(* CoDeSys 2.3.9.50 project: AXIS_CONTROL.pro *)
(* Libraries: TcBase.lib 14.5.09 12:14:08, TcSystem.lib 7.6.16 11:01:22, TcBaseMath.lib 27.7.04 12:07:56, TcMath.lib 23.9.04 15:15:30, TcNC.lib 10.10.08 17:55:34, TcUtilities.lib 3.2.16 16:08:58, TcEtherCAT.lib 30.11.16 19:52:18, TcTestAndSet.lib 23.2.09 12:50:08, TcDrive.lib 25.1.17 09:42:28, TcMc2Drive.lib 19.1.10 11:34:38, TcMC2.lib 19.10.15 15:49:44, STANDARD.LIB 5.6.98 12:03:02 *)

(* Task configuration *)
TASK Standard (PRIORITY := 0, INTERVAL := T#1ms);
	MAIN
END_TASK

(* Global variable list: Global_Variables_Hardware *)
VAR_GLOBAL

	input : STRING(35):='';
	Unit: REAL;
(*motor x*)
	fbNcAxis_Axis_X	: FB_NcAxis;
	stAxis_X			: ST_NcAxis;
	Axis_x			: AXIS_REF;


(*motor y*)
	fbNcAxis_Axis_Y	: FB_NcAxis;
	stAxis_Y			: ST_NcAxis;
	Axis_y			: AXIS_REF;

	Axis_dummy	: AXIS_REF;
END_VAR

(* Global variable list: TwinCAT_Configuration *)
(* Generated automatically by TwinCAT - (read only) *)
VAR_CONFIG
	.Axis_x.PlcToNc AT %QB0 : PLCTONC_AXIS_REF;	(*  ~ {LinkedWith:TINC^NC-Task 1 SAF^Axes^Axis 1^Inputs^Axis 1_FromPlc} *)
	.Axis_x.NcToPlc AT %IB0 : NCTOPLC_AXIS_REF;	(*  ~ {LinkedWith:TINC^NC-Task 1 SAF^Axes^Axis 1^Outputs^Axis 1_ToPlc} *)
	.Axis_y.PlcToNc AT %QB128 : PLCTONC_AXIS_REF;	(*  ~ {LinkedWith:TINC^NC-Task 1 SAF^Axes^Axis 2^Inputs^Axis 2_FromPlc} *)
	.Axis_y.NcToPlc AT %IB128 : NCTOPLC_AXIS_REF;	(*  ~ {LinkedWith:TINC^NC-Task 1 SAF^Axes^Axis 2^Outputs^Axis 2_ToPlc} *)
	.Axis_dummy.PlcToNc AT %QB256 : PLCTONC_AXIS_REF;
	.Axis_dummy.NcToPlc AT %IB256 : NCTOPLC_AXIS_REF;
END_VAR

(* Data type in DataTypes/FBsTypes/NC_Axis_Params/AxisVariables *)
TYPE ST_AxisVars :
STRUCT
	ax_ctrl:ST_ctrl;
	ax_stat:ST_stat;
END_STRUCT
END_TYPE

(* Data type in DataTypes/FBsTypes/NC_Axis_Params/AxisVariables *)
TYPE ST_ctrl :
STRUCT

(*ReadNCParam*)
	ReadParamExe:BOOL;
	ReadParamNum: mc_axisparameter:=AxisEncoderModuloValue;

(*Pwr,Reset*)
	Enable:BOOL;
	Enable_inhibit:BOOL;
	En_FW:BOOL;
	En_BW:BOOL;
	Reset:BOOL;
	Override:REAL:=100;
(*Stop*)
	StopExe:BOOL;
	StopDec:REAL;
(*SetPosition*)
	SetPosExe:BOOL;
	SetPosition:REAL;
(*Homing*)
	HomeExe:BOOL;
	HomeSW: BOOL;
	LimitSW_Max:BOOL;
	LimitSW_Min:BOOL;
	HomeSetPos:REAL;
	HomeOffsetPos:REAL;
	HomeOffsetVelo:REAL:=1;
(*Jog*)
	JogFW:BOOL;
	JogBW:BOOL;
	JogVel:REAL:=1;
	JogAcc:REAL;
	JogDec:REAL;
	JogMode: E_JogMode:=MC_JOGMODE_CONTINOUS;
(*MoveRelative*)
	MrelExe:BOOL;
	MrelDist:REAL;
	MrelVel:REAL:=1;
	MrelAcc:REAL;
	MrelDec:REAL;
(*MoveAbsolute*)
	MabsExe:BOOL;
	MabsPos:REAL;
	MabsVel:REAL:=1;
	MabsAcc:REAL;
	MabsDec:REAL;
	MabsBufferMode:MC_BufferMode;
(*MoveAbsoluteBlending*)
	MabsBlendExe:BOOL;
	MabsBlendPos:REAL;
	MabsBlendVel:REAL:=1;
	MabsBlendAcc:REAL;
	MabsBlendDec:REAL;
	MabsBlendBufferMode:MC_BufferMode;
(*MoveModulo*)
	MmodExe:BOOL;
	MmodPos:REAL;
	MmodVel:REAL:=1;
	MmodAcc:REAL;
	MmodDec:REAL;
	MmodDir:MC_Direction :=MC_Positive_Direction;(*MC_Positive_Direction := 1,MC_Shortest_Way ,MC_Negative_Direction ,  MC_Current_Direction *)
(*MoveVelocity*)
	MvelExe:BOOL;
	MvelVelo:REAL:=1;
	MvelAcc:REAL;
	MvelDec:REAL;
	MvelDirection:MC_Direction ;
	MvelPStopEnable:BOOL;
	MvelPStopPos:REAL;
	MvelPStopAcc:REAL;
	MvelPStopDec:REAL;
(*GearingDyn*)
	GrInDynExe:BOOL;
	GearRatio:REAL;
	GrInAcc:REAL;
	GrInDec:REAL;
	GearOut:BOOL;
(*GearingMultimaster*)
	GrInMMstrExe:BOOL;
	GearRatioMstr:REAL;
	GearRatioMstr2:REAL;
	GearRatioMstr3:REAL;
	GearRatioMstr4:REAL;
	GrInMMstrAcc:REAL;
	GrInMMstrDec:REAL;
	GearMMstrOut:BOOL;
(*TouchProbe*)
	TriggerRef : trigger_ref;
	TProbeExe:BOOL;
	TPWindowOnly: BOOL;
	TPFirstPosition:REAL;
	TPLastPosition :REAL;
(*AbortTouchProbe*)
	AbortTrigger:BOOL;
(*MoveSuperimposed*)
	SImpExe : 	BOOL;
	SImpMode : E_SuperpositionMode:=SUPERPOSITIONMODE_VELOREDUCTION_ADDITIVEMOTION;
	SImpDistance :REAL;
	SImpVelocityDiff :REAL;
	SImpAcc :REAL;
	SImpDec :REAL;
	SImpVelocityProcess :REAL;
	SImpLength :REAL;
	SImpOptions:ST_SuperpositionOptions;

(*ReadDiagnostics*)
	ExeDiagNumber:BOOL;
	cycDiagNumber:BOOL:=TRUE;
	ExeDiagNumberList       : BOOL;

(*ReadDiagMessage*)
	ExeReadDiagMessage:BOOL;
	cycReadDiagMessage:BOOL:=TRUE;









END_STRUCT
END_TYPE

(* Data type in NcAxisTypes/ST_NcAxisControl *)
TYPE ST_NcAxis :
STRUCT
	
	ctrl		: ST_NcAxisCtrl;
	stat		: ST_NcAxisStat;

END_STRUCT
END_TYPE

(* Data type in NcAxisTypes/ST_NcAxisControl/Sub_ST_NcAxis *)
TYPE ST_NcAxisCtrl :
STRUCT
	
(*ReadNCParam*)
	bReadNcParamExe:BOOL;
	eReadNcParamNum: mc_axisparameter:=AxisEncoderModuloValue;

	
(*WriteNCParam*)
	bWtiteNcParamExe:BOOL;
	eWriteNcParamNum: mc_axisparameter;
	fWriteNcParamValue:LREAL;


(*ReadDiagNumber*)
	bReadDiagNumber:BOOL;
	bReadDiagNumberCyc:BOOL:=TRUE;

	
(*ReadDiagNumberList*)
	bReadDiagNumberList:BOOL;

	
(*ReadDiagMessage*)
	bReadDiagMessage:BOOL;
	bReadDiagMessageCyc:BOOL:=TRUE;

	
(*McReset & SoeReset*)
	bReset:BOOL;
	bDriveReset:BOOL;
	bNcReset:BOOL;
	
	
(*Power*)
	bEnable:BOOL;
	bEnableInhibit:BOOL;
	bEnableBidirectional:BOOL:=TRUE;
	bEnablePositive:BOOL;
	bEnableNegative:BOOL;
	fOverride:REAL:=100;
	
	
(*Homing*)
	bHome:BOOL;
	bHomeSwitch: BOOL;
	fHomeSetPos:REAL;
	fHomeOffsetPos:REAL;
	fHomeOffsetVelo:REAL:=1;
	eHomingMode:MC_HomingMode:=MC_DefaultHoming;	
	(* 
		TYPE MC_HomingMode :
		(
			MC_DefaultHoming,    (* default homing as defined in the SystemManager encoder parameters *)
			MC_AbsSwitch,        (* not implemented - Absolute Switch homing plus Limit switches *)
			MC_LimitSwitch,      (* not implemented - Homing against Limit switches *)
			MC_RefPulse,         (* not implemented - Homing using encoder Reference Pulse "Zero Mark" *)
			MC_Direct,           (* Static Homing forcing position from user reference *)
			MC_Absolute,         (* not implemented - Static Homing forcing position from absolute encoder *)
			MC_Block,            (* not implemented - Homing against hardware parts blocking movement *)
			MC_ForceCalibration, (* set the calibration flag without perfomring any motion or changing the position *)
			MC_ResetCalibration  (* resets the calibration flag without perfomring any motion or changing the position *)
		);
		END_TYPE
	*)
	
	
(*Limit Switches*)
	bPositiveLimitSwitch:BOOL:=TRUE;
	bNegativeLimitSwitch:BOOL:=TRUE;
	
	
(*SetPosition*)
	bSetPosition:BOOL;
	fSetPosition:REAL;
	
	
(*Jog*)
	bJogForward:BOOL;
	bJogBackwards:BOOL;
	fJogPosition:REAL;
	fJogVelocity:REAL:=1;
	fJogAcc:REAL;
	fJogDec:REAL;
	eJogMode: E_JogMode:=MC_JOGMODE_CONTINOUS;
	(*
		TYPE E_JogMode :
		(
		   MC_JOGMODE_STANDARD_SLOW, (* motion with standard jog parameters for slow motion *)
		   MC_JOGMODE_STANDARD_FAST, (* motion with standard jog parameters for fast motion *)
		   MC_JOGMODE_CONTINOUS, (* axis moves as long as the jog button is pressed using parameterized dynamics *)
		   MC_JOGMODE_INCHING, (* axis moves for a certain relative distance *)
		   MC_JOGMODE_INCHING_MODULO (* axis moves for a certain relative distance - stop position is rounded to the distance value *)
		);
		END_TYPE
	*)
	
	
(*MoveRelative*)
	bMoveRelative:BOOL;
	fMoveRelDistance:LREAL;
	fMoveRelVelocity:REAL:=1;
	fMoveRelAcc:REAL;
	fMoveRelDec:REAL;
	eMoveRelBufferMode:MC_BufferMode;		

	
(*MoveAbsolute*)
	bMoveAbsolute:BOOL;
	fMoveAbsPosition:LREAL;
	fMoveAbsVelocity:REAL:=1;
	fMoveAbsAcc:REAL;
	fMoveAbsDec:REAL;
	eMoveAbsBufferMode:MC_BufferMode:=MC_Aborting;
	
	
(*MoveAbsoluteBlending*)
	bMoveAbsoluteBlending:BOOL;
	fMoveAbsBlendingPosition:LREAL;
	fMoveAbsBlendingVelocity:REAL:=1;
	fMoveAbsBlendingAcc:REAL;
	fMoveAbsBlendingDec:REAL;
	eMoveAbsBlendingBufferMode:MC_BufferMode:=MC_BlendingNext;
	(*
		TYPE MC_BufferMode :
		 (
		   MC_Aborting,
		   MC_Buffered,
		   MC_BlendingLow,
		   MC_BlendingPrevious,
		   MC_BlendingNext,
		   MC_BlendingHigh
		 );
		END_TYPE
	*)


(*MoveModulo*)
	bMoveModulo:BOOL;
	fMoveModuloPosition:LREAL;
	fMoveModuloVelocity:REAL:=1;
	fMoveModuloAcc:REAL;
	fMoveModuloDec:REAL;
	eMoveModuloBufferMode:MC_BufferMode;
	eMoveModuloDirection:MC_Direction :=MC_Positive_Direction;
	(*
		TYPE MC_Direction :
		(
		   MC_Positive_Direction := 1,
		   MC_Shortest_Way ,
		   MC_Negative_Direction,
		   MC_Current_Direction
		);
		END_TYPE 
	*)
	
	
(*MoveVelocity *)
	bMoveVelocity:BOOL;
	fMoveVelVelocity:REAL:=1;
	fMoveVelAcc:REAL;
	fMoveVelDec:REAL;
	eMoveVelDirection:MC_Direction ;
	eMoveVelBufferMode:MC_BufferMode:=MC_Aborting;
	(*Positional Stop *)
	bMoveVelPositionalStopEnable:BOOL;
	fMoveVelPositionalStopPos:REAL;
	(*fMoveVelPositionalStopVelo:REAL;*)
	fMoveVelPositionalStopAcc:REAL;
	fMoveVelPositionalStopDec:REAL;
	eMoveVelPositionalStopBufferMode:MC_BufferMode:=MC_BlendingNext;


(*Gearing Dynamic Axis1 to Master *)
	bGearInDynamic_Axis1toMaster:BOOL;
	fGearInDynRatio_Axis1toMaster:REAL;
	fGearInDynAcc_Axis1toMaster:REAL;
	fGearInDynDec_Axis1toMaster:REAL;
	
	
(*Gearing Dynamic *)
	bGearInDynamic:BOOL;
	fGearInDynRatio:REAL;
	fGearInDynAcc:REAL;
	fGearInDynDec:REAL;
	
	
(*GearingMultimaster*)
	bGearInMultimaster:BOOL;
	fGearRatioMaster1:REAL;
	fGearRatioMaster2:REAL;
	fGearRatioMaster3:REAL;
	fGearRatioMaster4:REAL;
	fGearInMultimasterAcc:REAL;
	fGearInMultimasterDec:REAL;
	
	
(*MoveSuperimposed*)
	bMoveSuperimposed:BOOL;
	fMoveSupImpDistance:LREAL;
	fMoveSupImpVelocityDiff:REAL;
	fMoveSupImpAcc:REAL;
	fMoveSupImpDec:REAL;
	fMoveSupImpVelocityProcess:REAL;
	fMoveSupImpLength:REAL;
	eMoveSupImpOptions:ST_SuperpositionOptions;
	(*
		TYPE ST_SuperpositionOptions :
		STRUCT
		   AbortOption : E_SuperpositionAbortOption;
		END_STRUCT
		END_TYPE 
		 
		TYPE E_SuperpositionAbortOption :
		 (
			SUPERPOSITIONOPTION_ABORTATSTANDSTILL := 0, 
			SUPERPOSITIONOPTION_RESUMEAFTERSTANDSTILL, 
			SUPERPOSITIONOPTION_RESUMEAFTERMOTIONSTOP 
		 );
		END_TYPE 
	*)
	
	eMoveSupImpMode:E_SuperpositionMode:=SUPERPOSITIONMODE_VELOREDUCTION_ADDITIVEMOTION;
	(*
		TYPE E_SuperpositionMode :
		(
		 SUPERPOSITIONMODE_VELOREDUCTION_ADDITIVEMOTION := 1,
		 SUPERPOSITIONMODE_VELOREDUCTION_LIMITEDMOTION,
		 SUPERPOSITIONMODE_LENGTHREDUCTION_ADDITIVEMOTION,
		 SUPERPOSITIONMODE_LENGTHREDUCTION_LIMITEDMOTION,
		 SUPERPOSITIONMODE_ACCREDUCTION_ADDITIVEMOTION, (from TwinCAT
		2.11)
		 SUPERPOSITIONMODE_ACCREDUCTION_LIMITEDMOTION (from TwinCAT
		2.11)
		);
		END_TYPE 
	*)

	
(*Gear Out*)
	bGearOutSlaveAxis:BOOL;
	
	
(*Gear Out*)
	bGearOutAxis1fromMaster:BOOL;
	
	
(*TouchProbe*)
	bTouchProbe:BOOL;
	bTouchProbeWindowOnly:BOOL;
	fTouchProbeFirstPosition:LREAL;
	fTouchProbeLastPosition:LREAL;
	eTouchProbeTriggerRef:trigger_ref;
	
	
(*AbortTouchProbe*)
	bTouchProbeAbortTrigger:BOOL;
	
	
(*Stop Axis1*)
	bStopAxis:BOOL;
	fStopAxisDec:REAL;
	
		
(*External Setposition Generation*)
	bExtSetPointGenEnable:BOOL;
	fExtSetPosition:LREAL;
	fExtSetVelocity:LREAL;
	fExtSetAcceleration:LREAL;
	iExtSetDirection:DINT;
	eExtSetPositionType: E_POSITIONTYPE :=POSITIONTYPE_ABSOLUTE; 
	 (*
		TYPE E_PositionType :
		(
		   POSITIONTYPE_ABSOLUTE  := 1, (* Absolute position *)
		   POSITIONTYPE_RELATIVE,       (* Relative position *)
		   POSITIONTYPE_MODULO    := 5  (* Modulo position *)
		);
		END_TYPE
	*)

	
END_STRUCT
END_TYPE

(* Data type in NcAxisTypes/ST_NcAxisControl/Sub_ST_NcAxis *)
TYPE ST_NcAxisStat :
STRUCT
	
(*ReadNCParam*)
	bReadNcParamValid:BOOL;
	bReadNcParamBusy:BOOL;
	bReadNcParamError:BOOL;
	iReadNcParamErrID:UDINT;
	fReadNcParamValue:LREAL;
	
	
(*MaxVelo & Modulo*)
	bMaxVeloModuloinitialized:BOOL;
	fModuloValue:LREAL;
	fMaxVelocity:LREAL;
	
	
(*WriteNCParam*)
	bWriteNcParamDone:BOOL;
	bWriteNcParamBusy:BOOL;
	bWriteNcParamError:BOOL;
	iWriteNcParamErrID:UDINT;
	

(*Status, Power, Reset*)
	bAxisError:BOOL;
	iAxisErrID:UDINT;
	
	
(*ReadDiagNumber*)
	bReadDiagNumberBusy:BOOL;
	bReadDiagNumberError:BOOL;
	iReadDiagNumberAdsErrId:UINT;
	iReadDiagNumberSercosErrId:UINT;
	iReadDiagNumber:UDINT;
	iReadDiagNumberAttribute:DWORD;
	
	
(*ReadDiagNumberlist*)
	stReadDiagNumberList:ST_SoE_DiagNumList;
	bReadDiagNumberListBusy:BOOL;
	bReadDiagNumberListError:BOOL;
	iReadDiagNumberListAdsErrId:UINT;
	iReadDiagNumberListSercosErrId:UINT;
	iReadDiagNumberListAttribute:DWORD;
	
	
(*ReadDiagMessage*)
	bReadDiagMessageBusy:BOOL;
	bReadDiagMessageError:BOOL;
	iReadDiagMessageAdsErrId:UINT;
	iReadDiagMessageSercosErrId:UINT;
	sReadDiagMessage:ST_Soe_String;
	iReadDiagMessageAttribute:DWORD;
	
	
(*Reset*)
	bResetDone:BOOL;
	bResetBusy:BOOL;
	bResetError:BOOL;
	iResetErrID:UDINT;

	bSoeResetDone:BOOL;
	bSoeResetBusy:BOOL;
	bSoeResetError:BOOL;
	iSoeResetErrID:UDINT;
	iSoeResetSercosErrID:UDINT;
	
	
(*Power*)
	bPowered:BOOL;
	bPowerBusy:BOOL;
	bPowerActive:BOOL;
	bPowerError:BOOL;
	iPowerErrID:UDINT;
	
	
(*Homing*)
	bHomeDone:BOOL;
	bHomeBusy:BOOL;
	bHomeActive:BOOL;
	bHomeAborted:BOOL;
	bHomeError:BOOL;
	iHomeErrID:UDINT;

	bHomeOffsDone:BOOL;
	bHomeOffsBusy:BOOL;	
	bHomeOffsActive:BOOL;
	bHomeOffsAborted:BOOL;
	bHomeOffsError:BOOL;
	iHomeOffsErrID:UDINT;
	
	bHomed:BOOL;
	
	
(*SetPosition*)
	bSetPositionDone:BOOL;
	bSetPositionBusy:BOOL;
	bSetPositionError:BOOL;
	iSetPositionErrID:UDINT;
	
	
(*Jog*)
	bJogDone:BOOL;
	bJogBusy:BOOL;
	bJogActive:BOOL;
	bJogAborted:BOOL;
	bJogError:BOOL;
	iJogErrID:UDINT;
	
	
(*MoveRelative*)
	bMoveRelDone:BOOL;
	bMoveRelBusy:BOOL;
	bMoveRelActive:BOOL;
	bMoveRelAborted:BOOL;
	bMoveRelErr:BOOL;
	iMoveRelErrID:UDINT;
		
	
(*MoveAbsolute*)
	bMoveAbsDone:BOOL;
	bMoveAbsBusy:BOOL;
	bMoveAbsActive:BOOL;
	bMoveAbsAborted:BOOL;
	bMoveAbsErr:BOOL;
	iMoveAbsErrID:UDINT;

	
(*MoveAbsoluteBlending*)
	bMoveAbsBlendingDone:BOOL;
	bMoveAbsBlendingBusy:BOOL;
	bMoveAbsBlendingActive:BOOL;
	bMoveAbsBlendingAborted:BOOL;
	bMoveAbsBlendingErr:BOOL;
	iMoveAbsBlendingErrID:UDINT;
	
	
(*MoveModulo*)
	bMoveModuloDone:BOOL;
	bMoveModuloBusy:BOOL;
	bMoveModuloActive:BOOL;
	bMoveModuloAborted:BOOL;
	bMoveModuloErr:BOOL;
	iMoveModuloErrID:UDINT;	

	
(*MoveVelocity *)
	bMoveVeloInVelocity:BOOL;
	bMoveVeloBusy:BOOL;
	bMoveVeloActive:BOOL;
	bMoveVeloAborted:BOOL;
	bMoveVeloErr:BOOL;
	iMoveVeloErrID:UDINT;
	(*Positional Stop *)
	bMoveVeloPosStopDone:BOOL;
	bMoveVeloPosStopBusy:BOOL;
	bMoveVeloPosStopActive:BOOL;
	bMoveVeloPosStopAborted:BOOL;
	bMoveVeloPosStopErr:BOOL;
	iMoveVeloPosStopErrID:UDINT;
	
	
(*Gearing Dynamic *)
	bGearInDynInGear:BOOL;
	bGearInDynBusy:BOOL;
	bGearInDynActive:BOOL;
	bGearInDynAborted:BOOL;
	bGearInDynErr:BOOL;
	iGearInDynErrID:UDINT;
	
	
(*Gearing Dynamic Axis1 to Master *)	
	bGearInDynInGear_Axis1toMaster:BOOL;
	bGearInDynBusy_Axis1toMaster:BOOL;
	bGearInDynActive_Axis1toMaster:BOOL;
	bGearInDynAborted_Axis1toMaster:BOOL;
	bGearInDynErr_Axis1toMaster:BOOL;
	iGearInDynErrID_Axis1toMaster:UDINT;	
	
	
(*Gearing Multimaster*)
	bGearInMultimasterInGear:BOOL;
	bGearInMultimasterBusy:BOOL;
	bGearInMultimasterActive:BOOL;
	bGearInMultimasterAborted:BOOL;
	bGearInMultimasterErr:BOOL;
	iGearInMultimasterGrErrID:UDINT;	
	
	
(*MoveSuperimposed*)
	bMoveSupImpDone:BOOL;
	bMoveSupImpBusy:BOOL;
	bMoveSupImpActive:BOOL;
	bMoveSupImpAborted:BOOL;
	bMoveSupImpErr:BOOL;
	iMoveSupImpErrorId:UDINT;
	bMoveSupImpWarning:BOOL;
	iMoveSupImpWarningID:UDINT;
	fMoveSupImpActualVelocityDiff:LREAL;
	fMoveSupImpActualDistance:LREAL;
	fMoveSupImpActualLength:LREAL;
	fMoveSupImpActualAcc:LREAL;
	fMoveSupImpActualDec:LREAL;	

	
(*Gear Out*)
	bGearOutSlaveAxisDone:BOOL;
	bGearOutSlaveAxisBusy:BOOL;
	bGearOutSlaveAxisErr:BOOL;
	iGearOutSlaveAxisErrID:UDINT;
	
	
(*Gear Out Axis1 from Master*)
	bGearOutAxis1fromMasterDone:BOOL;
	bGearOutAxis1fromMasterBusy:BOOL;
	bGearOutAxis1fromMasterErr:BOOL;
	iGearOutAxis1fromMasterErrID:UDINT;

	
(*SlaveStop*)
	bStopSlaveAxisDone:BOOL;
	bStopSlaveAxisBusy:BOOL;
	bStopSlaveAxisActive:BOOL;
	bStopSlaveAxisAborted:BOOL;
	bStopSlaveAxisErr:BOOL;
	iStopSlaveAxisErrorID:UDINT;
	
	
(*TouchProbe*)
	bTouchProbeDone:BOOL;
	bTouchProbeBusy:BOOL;
	bTouchProbeAborted:BOOL;
	bTouchProbeErr:BOOL;
	iTouchProbeErrID:UDINT;
	fTouchProbeRecordedPosition:LREAL;
	eTouchProbeRecordedData:MC_TouchProbeRecordedData; 	
	(*
		TYPE MC_TouchProbeRecordedData :
		STRUCT
			Counter             : LREAL;
			RecordedPosition    : LREAL;
			AbsolutePosition    : LREAL;
			ModuloPosition      : LREAL;
		END_STRUCT
		END_TYPE
	*)
	
	
(*AbortTouchProbe*)
	bAbortTouchProbeDone:BOOL;
	bAbortTouchProbeBusy:BOOL;
	bAbortTouchProbeErr:BOOL;
	iAbortTouchProbeErrID:UDINT;
	
	
(*Stop Axis1*)
	bStopAxisDone:BOOL;
	bStopAxisBusy:BOOL;
	bStopAxisActive:BOOL;
	bStopAxisAborted:BOOL;
	bStopAxisErr:BOOL;
	iStopAxisErrID:UDINT;
	
	
(*External Setposition Generation*)
	bExtSetPositionReady:BOOL;
	bExtSetPositionDone:BOOL;
	bExtSetPositionBusy:BOOL;
	bExtSetPositionErr:BOOL;
	iExtSetPositionErrID:UDINT;


END_STRUCT
END_TYPE

(* Data type in DataTypes/FBsTypes/NC_Axis_Params/AxisVariables *)
TYPE ST_stat :
STRUCT
(*ReadNCParam*)
	ReadParamValid:BOOL;
	ReadParamBusy:BOOL;
	ReadParamError:BOOL;
	ReadParamErrID:UDINT;
	ReadParamValue:LREAL;

	ModuloValue:LREAL;
	MaxVelocity:REAL;

(*Pwr,Reset*)
	ResetDone:BOOL;
	ResetBusy:BOOL;
	ResetError:BOOL;
	ResetErrID:UDINT;

	SoeResetDone:BOOL;
	SoeResetBusy:BOOL;
	SoeResetError:BOOL;
	SoeResetErrID:UDINT;

	AxisError:BOOL;
	AxisErrID:UDINT;

	Powered:BOOL;
	PowBusy:BOOL;
	PowActive:BOOL;
	PowError:BOOL;
	PowErrID:UDINT;
(*Stop*)
	StopDone : BOOL;
	StopBusy : BOOL;
	StopActive : BOOL;
	StopCommandAborted: BOOL;
	StopError : BOOL;
	StopErrorID : UDINT;
(*SlaveStop*)
	SlaveStopDone : BOOL;
	SlaveStopBusy : BOOL;
	SlaveStopActive : BOOL;
	SlaveStopCommandAborted: BOOL;
	SlaveStopError : BOOL;
	SlaveStopErrorID : UDINT;
(*SetPosition*)
	SetPosDone:BOOL;
	SetPosBusy:BOOL;
	SetPosError:BOOL;
	SetPosErrID:UDINT;
(*Homing*)
	HomeDone:BOOL;
	Homed:BOOL;
	HomeError:BOOL;
	HomeErrID:UDINT;
	HomeOffsDone:BOOL;
	HomeOffsBusy:BOOL;
	HomeOffsError:BOOL;
	HomeOffsErrID:UDINT;
(*Jog*)
	JogBusy:BOOL;
	JogError:BOOL;
(*MoveRelative*)
	MrelDone:BOOL;
	MrelBusy:BOOL;
	MrelAborted:BOOL;
	MrelErr:BOOL;
	MrelErrID:UDINT;
(*MoveAbsolute*)
	MabsDone:BOOL;
	MabsBusy:BOOL;
	MabsAborted:BOOL;
	MabsErr:BOOL;
	MabsErrID:UDINT;
(*MoveAbsoluteBlending*)
	MabsBlendDone:BOOL;
	MabsBlendBusy:BOOL;
	MabsBlendAborted:BOOL;
	MabsBlendErr:BOOL;
	MabsBlendErrID:UDINT;
(*MoveModulo*)
	MmodDone:BOOL;
	MmodBusy:BOOL;
	MmodAborted:BOOL;
	MmodErr:BOOL;
	MmodErrID:UDINT;
(*MoveVelocity*)
	MvelinVelo:BOOL;
	MvelBusy:BOOL;
	MvelAborted:BOOL;
	MvelErr:BOOL;
	MvelErrID:UDINT;
	MvelPStopDone:BOOL;
	MvelPStopBusy:BOOL;
	MvelPStopActive:BOOL;
	MvelPStopComAborted:BOOL;
	MvelPStopError:BOOL;
	MvelPStopErrID:UDINT;
(*GearingDyn*)
	InGear:BOOL;
	GrInBusy:BOOL;
	GrInAborted:BOOL;
	GrError:BOOL;
	GrErrID:UDINT;
	GrOutDone:BOOL;
	GrOutBusy:BOOL;
	GrOutError:BOOL;
	GrOutErrID:UDINT;
(*GearingMMstr*)
	InGear_MMstr:BOOL;
	GrInBusy_MMstr:BOOL;
	GrInActive_MMstr:BOOL;
	GrInAborted_MMstr:BOOL;
	GrError_MMstr:BOOL;
	GrErrID_MMstr:UDINT;
(*TouchProbe*)
	TPDone: BOOL;
	TPBusy: BOOL;
	TPCommandAborted: BOOL;
	TPError: BOOL;
	TPErrorID: UDINT;
	TPRecordedPosition: REAL;
(*AbortTouchProbe*)
	AbortTP_Done : BOOL;
	AbortTP_Busy : BOOL;
	AbortTP_Error : BOOL;
	AbortTP_ErrorID : UDINT;
(*MoveSuperimposed*)
	SImpDone: BOOL;
	SImpBusy : BOOL;
	SImpActive : BOOL;
	SImpCommandAborted : BOOL;
	SImpError : BOOL;
	SImpErrorId : UDINT;
	SImpWarning : BOOL;
	SImpWarningID : UDINT;
	SImpActualVelocityDiff	:REAL;
	SImpActualDistance :REAL;
	SImpActualLength 	:REAL;
	SImpActualAcceleration : REAL;
	SImpActualDeceleration : REAL;
(*ReadDiagnostics*)
	DiagBusy: BOOL;
	DiagError: BOOL;
	DiagAdsErrId: UINT;
	DiagSercosErrId: UINT;
	DiagNumber:UDINT;
	DiagAttribute:DWORD;
(*ReadDiaglist*)
	stDiagNumberList:ST_SoE_DiagNumList;
	DiagListBusy:BOOL;
	DiagListError:BOOL;
	DiagListAdsErrId:UINT;
	DiagListSercosErrId:UINT;
	DiagListAttribute:DWORD;

(*ReadDiagMessage*)
	ReadDiagMessageBusy: BOOL;
	ReadDiagMessageError: BOOL;
	ReadDiagMessageAdsErrId: UINT;
	ReadDiagMessageSercosErrId:UINT;
	ReadDiagMessage:ST_Soe_String;
	ReadDiagMessageAttribute:DWORD;


END_STRUCT
END_TYPE

(* POU MAIN, LD *)
PROGRAM MAIN
VAR
	prefExtSetPosition: REAL;

	fCounter: REAL;
	bStart: BOOL;

END_VAR
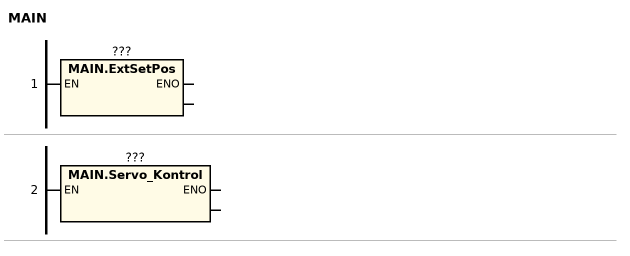
_LD_ (* Ladder Diagram *)
NETWORK 1
	*
		EN --- ???:MAIN.ExtSetPos()
NETWORK 2
	*
		EN --- ???:MAIN.Servo_Kontrol()
_END_LD_
END_PROGRAM
ACTION ExtSetPos:
	Unit;
	input;
	(*input := TRUNC(fUnit);*)
	Unit :=STRING_TO_REAL(input);

	IF bStart THEN

		stAxis_X.ctrl.bEnable:=TRUE;

		IF stAxis_x.stat.bPowered THEN

			stAxis_X.ctrl.bExtSetPointGenEnable :=stAxis_x.stat.bPowered;

			stAxis_X.ctrl.fExtSetPosition		:= Unit;
			stAxis_X.ctrl.fExtSetVelocity		:= (stAxis_X.ctrl.fExtSetPosition-prefExtSetPosition)/(0.01);
			stAxis_X.ctrl.fExtSetAcceleration;

			IF stAxis_X.ctrl.fExtSetVelocity>0 THEN
				stAxis_X.ctrl.iExtSetDirection :=1;

			ELSIF stAxis_X.ctrl.fExtSetVelocity<0 THEN
				stAxis_X.ctrl.iExtSetDirection :=(-1);

			ELSE
				stAxis_X.ctrl.iExtSetDirection :=0;
			END_IF
		
			prefExtSetPosition :=stAxis_X.ctrl.fExtSetPosition;
		
			stAxis_X.stat.bExtSetPositionReady;
	
		END_IF

	ELSE
		stAxis_X.ctrl.bEnable:=FALSE;
		stAxis_X.ctrl.bExtSetPointGenEnable :=stAxis_x.stat.bPowered;
	END_IF
END_ACTION
ACTION Servo_Kontrol:
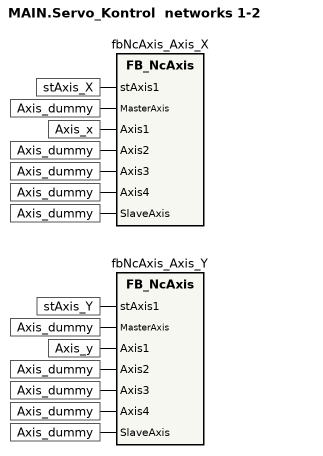
_FBD_ (* Function Block Diagram *)
NETWORK 1
	fbNcAxis_Axis_X:FB_NcAxis(stAxis1: stAxis_X, MasterAxis: Axis_dummy, Axis1: Axis_x, Axis2: Axis_dummy, Axis3: Axis_dummy, Axis4: Axis_dummy, SlaveAxis: Axis_dummy)
NETWORK 2
	fbNcAxis_Axis_Y:FB_NcAxis(stAxis1: stAxis_Y, MasterAxis: Axis_dummy, Axis1: Axis_y, Axis2: Axis_dummy, Axis3: Axis_dummy, Axis4: Axis_dummy, SlaveAxis: Axis_dummy)
_END_FBD_
(* the same logic as Structured Text *)
(* Network 1 *)
fbNcAxis_Axis_X(stAxis1 := stAxis_X, MasterAxis := Axis_dummy, Axis1 := Axis_x, Axis2 := Axis_dummy, Axis3 := Axis_dummy, Axis4 := Axis_dummy, SlaveAxis := Axis_dummy);
(* Network 2 *)
fbNcAxis_Axis_Y(stAxis1 := stAxis_Y, MasterAxis := Axis_dummy, Axis1 := Axis_y, Axis2 := Axis_dummy, Axis3 := Axis_dummy, Axis4 := Axis_dummy, SlaveAxis := Axis_dummy);
END_ACTION

(* POU FBs/FB_NcAxis, ST *)
FUNCTION_BLOCK FB_NcAxis

VAR_INPUT
END_VAR

VAR_OUTPUT
END_VAR

VAR
	fbReadParameter: MC_ReadParameter;
	fbWriteParameter: MC_WriteParameter;
	iniReadMaxVeloModuloSTATE: INT;
	tonRetryReadMaxVeloModulo: TON;
	fbReadStatus: MC_ReadStatus;
	fbSoEReadDiagNumber: FB_SoEReadDiagNumber;
	fbSoEReadDiagNumberList: FB_SoEReadDiagNumberList;
	fbSoEReadDiagMessage: FB_SoEReadDiagMessage;
	fbReset: MC_Reset;
	fbSoEReset: FB_SoEReset;
	bDriveError: BOOL;
	fbPower: MC_Power;
	fbHome: MC_Home;
	fbMoveAbsoluteHomeOffs: MC_MoveAbsolute;
	RebHome: R_TRIG;
	fbSetPosition: MC_SetPosition;
	fbJog: MC_Jog;
	fbMoveRelative: MC_MoveRelative;
	fbMoveAbsolute: MC_MoveAbsolute;
	fbMoveAbsoluteBlending: MC_MoveAbsolute;
	fbMoveModulo: MC_MoveModulo;
	fbMoveVelocity: MC_MoveVelocity;
	ReMoveVelocity: R_TRIG;
	FeMoveVelocity: F_TRIG;
	oldMoveVeloVelocity: REAL;
	oldDirection: MC_Direction;
	bMoveVelocity: BOOL;
	fbMoveVeloPosStop: MC_MoveAbsolute;
	bStopAxis1: BOOL;
	fbGearInDyn: MC_GearInDyn;
	fbGearInDyn_Axis1toMaster: MC_GearInDyn;
	fbGearInMultiMaster: MC_GearInMultiMaster;
	fbMoveSuperImposed: MC_MoveSuperImposed;
	fbGearOut: MC_GearOut;
	fbGearOutAxis1fromMaster: MC_GearOut;
	fbStopSlave: MC_Stop;
	fbTouchProbe: MC_TouchProbe;
	fbAbortTrigger: MC_AbortTrigger;
	fbStopMaster: MC_Stop;
	
	ExtSP_State: INT;
	preExtSP_State: INT;
	fbExtSetPointGenEnable: MC_ExtSetPointGenEnable;
	fbExtSetPointGenDisable: MC_ExtSetPointGenDisable;
END_VAR


VAR_IN_OUT
	stAxis1:ST_NcAxis;
	MasterAxis:AXIS_REF;
	Axis1:AXIS_REF;
	Axis2:AXIS_REF;
	Axis3:AXIS_REF;
	Axis4:AXIS_REF;
	SlaveAxis:AXIS_REF;
END_VAR
(*Read Axis Parameter *)
	
	fbReadParameter(
		Axis			:= Axis1,
		Enable			:= stAxis1.ctrl.bReadNcParamExe, 
		ParameterNumber	:= stAxis1.ctrl.eReadNcParamNum, 
		ReadMode		:= READMODE_ONCE, 
		Valid			=> stAxis1.stat.bReadNcParamValid, 
		Busy			=> stAxis1.stat.bReadNcParamBusy, 
		Error			=> stAxis1.stat.bReadNcParamError, 
		ErrorID			=> stAxis1.stat.iReadNcParamErrID, 
		Value			=> stAxis1.stat.fReadNcParamValue );
		
		
(*Write Axis Parameter *)
	
	fbWriteParameter(
		Axis			:= Axis1, 
		Execute			:= stAxis1.ctrl.bWtiteNcParamExe, 
		ParameterNumber	:= stAxis1.ctrl.eWriteNcParamNum, 
		Value			:= stAxis1.ctrl.fWriteNcParamValue, 
		Done			=> stAxis1.stat.bWriteNcParamDone, 
		Busy			=> stAxis1.stat.bWriteNcParamBusy, 
		Error			=> stAxis1.stat.bWriteNcParamError, 
		ErrorID			=> stAxis1.stat.iWriteNcParamErrID );
		
		
		
(*initial reading of Modulo & MaxVelo ************************************************)		
		
	CASE iniReadMaxVeloModuloSTATE OF
		0:	
			IF NOT(stAxis1.stat.bMaxVeloModuloinitialized) THEN
				iniReadMaxVeloModuloSTATE:=10;
			END_IF
	
		10:
			stAxis1.ctrl.eReadNcParamNum:=AxisEncoderModuloValue;
			stAxis1.ctrl.bReadNcParamExe:=TRUE;
	
			iniReadMaxVeloModuloSTATE:=20;
			
		20:
			IF NOT(stAxis1.stat.bReadNcParamError) THEN
				IF NOT(stAxis1.stat.bReadNcParamBusy) THEN
					stAxis1.stat.fModuloValue:=stAxis1.stat.fReadNcParamValue;
					stAxis1.ctrl.bReadNcParamExe:=FALSE;
					iniReadMaxVeloModuloSTATE:=30;
				END_IF			
			ELSE
				iniReadMaxVeloModuloSTATE:=99;
			END_IF
	
		30:	
			stAxis1.ctrl.eReadNcParamNum:=AxisVeloMax;
			stAxis1.ctrl.bReadNcParamExe:=TRUE;
	
			iniReadMaxVeloModuloSTATE:=40;
			
		40:	
			IF NOT(stAxis1.stat.bReadNcParamError) THEN
				IF NOT(stAxis1.stat.bReadNcParamBusy) THEN
					stAxis1.stat.fMaxVelocity:=stAxis1.stat.fReadNcParamValue;
					stAxis1.ctrl.bReadNcParamExe:=FALSE;
					iniReadMaxVeloModuloSTATE:=50;
				END_IF			
			ELSE
				iniReadMaxVeloModuloSTATE:=99;
			END_IF
		
		50:(*MaxVelo & Modulo initialized*)
			stAxis1.stat.bMaxVeloModuloinitialized:=TRUE;
		
		99:(*error*)
			stAxis1.ctrl.bReadNcParamExe:=FALSE;
			tonRetryReadMaxVeloModulo(IN:=TRUE , PT:=T#3S , Q=> , ET=> );
			IF tonRetryReadMaxVeloModulo.Q THEN
				iniReadMaxVeloModuloSTATE:=0;
			END_IF
	END_CASE
	
(*initial reading of Modulo & MaxVelo ///////////////////////////////////////////////*)		



(*Read Status *)
		Axis1.ReadStatus();
		stAxis1.stat.bAxisError:=Axis1.Status.Error;
		stAxis1.stat.iAxisErrID:=Axis1.Status.ErrorID;
		
			
(*Read DiagNumber *)
	fbSoEReadDiagNumber(
		NetId:= '', 
		Execute:= stAxis1.ctrl.bReadDiagNumber OR (stAxis1.ctrl.bReadDiagNumberCyc AND NOT(stAxis1.stat.bReadDiagNumberBusy)), 
		Timeout:= T#2S, 
		Axis:= Axis1, 
		Busy=> stAxis1.stat.bReadDiagNumberBusy, 
		Error=> stAxis1.stat.bReadDiagMessageError, 
		AdsErrId=> stAxis1.stat.iReadDiagNumberAdsErrId, 
		SercosErrId=> stAxis1.stat.iReadDiagMessageSercosErrId, 
		DiagNumber=> stAxis1.stat.iReadDiagNumber, 
		Attribute=> stAxis1.stat.iReadDiagNumberAttribute );		


(*Read DiagNumberList *)
	fbSoEReadDiagNumberList(
		NetId:= '', 
		Execute:= stAxis1.ctrl.bReadDiagNumberList, 
		Timeout:= T#4S, 
		pDiagNumber:= ADR(stAxis1.stat.stReadDiagNumberList), 
		Size:= SIZEOF(stAxis1.stat.stReadDiagNumberList), 
		Axis:= Axis1, 
		Busy=> stAxis1.stat.bReadDiagNumberListBusy, 
		Error=> stAxis1.stat.bReadDiagNumberListError, 
		AdsErrId=> stAxis1.stat.iReadDiagNumberListAdsErrId, 
		SercosErrId=> stAxis1.stat.iReadDiagMessageSercosErrId, 
		Attribute=> stAxis1.stat.iReadDiagNumberListAttribute );
		

(*Read DiagMessage *)
	fbSoEReadDiagMessage(
		NetId:= '', 
		Execute:= stAxis1.ctrl.bReadDiagMessage OR (stAxis1.ctrl.bReadDiagMessageCyc AND NOT(stAxis1.stat.bReadDiagMessageBusy)), 
		Timeout:= T#2S, 
		Axis:= Axis1, 
		Busy=> stAxis1.stat.bReadDiagMessageBusy, 
		Error=> stAxis1.stat.bReadDiagMessageError, 
		AdsErrId=> stAxis1.stat.iReadDiagMessageAdsErrId, 
		SercosErrId=> stAxis1.stat.iReadDiagMessageSercosErrId, 
		DiagMessage=> stAxis1.stat.sReadDiagMessage, 
		Attribute=> stAxis1.stat.iReadDiagMessageAttribute );
	

(*NC Reset *)		
	fbReset(
		Axis:= Axis1, 
		Execute:= stAxis1.ctrl.bNcReset OR (stAxis1.ctrl.bReset AND Axis1.Status.Error AND NOT(stAxis1.stat.bResetError)), 
		Done=> stAxis1.stat.bResetDone, 
		Busy=> stAxis1.stat.bResetBusy, 
		Error=> stAxis1.stat.bResetError, 
		ErrorID=> stAxis1.stat.iResetErrID );
	

(*Drive SoeReset *)			
	bDriveError:=(stAxis1.stat.iReadDiagNumber<>16#D011 OR stAxis1.stat.iReadDiagNumber<>16#D012 OR stAxis1.stat.iReadDiagNumber<>16#D013);
	
	fbSoEReset(
		NetId:= '', 
		Execute:= stAxis1.ctrl.bDriveReset OR (stAxis1.ctrl.bReset AND (Axis1.Status.Error OR bDriveError)), 
		Timeout:= T#2S, 
		Axis:= Axis1, 
		Busy=> stAxis1.stat.bSoeResetBusy,
		Error=> stAxis1.stat.bSoeResetError, 
		AdsErrId=> stAxis1.stat.iSoeResetErrID, 
		SercosErrId=> stAxis1.stat.iSoeResetSercosErrID );
		

(*Power *)
	IF stAxis1.ctrl.bEnableBidirectional THEN
		stAxis1.ctrl.bEnablePositive:=stAxis1.ctrl.bEnable;
		stAxis1.ctrl.bEnableNegative:=stAxis1.ctrl.bEnable;
	ELSE
		;
	END_IF

	fbPower(
		Axis:= Axis1,
		Enable:= stAxis1.ctrl.bEnable AND NOT(stAxis1.stat.bAxisError OR stAxis1.ctrl.bEnableInhibit), 
		Enable_Positive:= stAxis1.ctrl.bEnablePositive AND NOT(stAxis1.stat.bAxisError OR stAxis1.ctrl.bEnableInhibit), 
		Enable_Negative:= stAxis1.ctrl.bEnableNegative AND NOT(stAxis1.stat.bAxisError OR stAxis1.ctrl.bEnableInhibit), 
		Override:= stAxis1.ctrl.fOverride, 
		BufferMode:= ,
		Status=> stAxis1.stat.bPowered, 
		Busy=> stAxis1.stat.bPowerBusy, 
		Active=> stAxis1.stat.bPowerActive, 
		Error=> stAxis1.stat.bPowerError, 
		ErrorID=> stAxis1.stat.iPowerErrID );



(*Homing *)	
	fbHome(
		Axis:= Axis1,
		Execute:= (stAxis1.ctrl.bHome AND stAxis1.stat.bPowered), 
		Position:= stAxis1.ctrl.fHomeSetPos, 
		HomingMode:= stAxis1.ctrl.eHomingMode, 
		BufferMode:= , 
		Options:= , 
		bCalibrationCam:= stAxis1.ctrl.bHomeSwitch, 
		Done=> stAxis1.stat.bHomeDone, 
		Busy=> stAxis1.stat.bHomeBusy, 
		Active=> stAxis1.stat.bHomeActive, 
		CommandAborted=> stAxis1.stat.bHomeAborted, 
		Error=> stAxis1.stat.bHomeError, 
		ErrorID=> stAxis1.stat.iHomeErrID );

	
	fbMoveAbsoluteHomeOffs(
		Axis:= Axis1, 
		Execute:= stAxis1.stat.bHomeDone, 
		Position:= stAxis1.ctrl.fHomeOffsetPos, 
		Velocity:= stAxis1.ctrl.fHomeOffsetVelo, 
		Acceleration:= , 
		Deceleration:= , 
		Jerk:= , 
		BufferMode:= , 
		Options:= , 
		Done=> stAxis1.stat.bHomeOffsDone, 
		Busy=> stAxis1.stat.bHomeOffsBusy, 
		Active=> stAxis1.stat.bHomeOffsActive, 
		CommandAborted=> stAxis1.stat.bHomeOffsAborted, 
		Error=> stAxis1.stat.bHomeOffsError, 
		ErrorID=> stAxis1.stat.iHomeOffsErrID);		
		
		
	RebHome(CLK:=stAxis1.ctrl.bHome , Q=> );
	
	IF RebHome.Q OR NOT(Axis1.Status.Homed) THEN
		stAxis1.stat.bHomed:=FALSE;
	ELSIF stAxis1.stat.bHomeOffsDone THEN
		stAxis1.stat.bHomed:=TRUE;
	END_IF
		
	
(*Hard Limit Switches *)
	Axis1.PlcToNc.ControlDWord:=AxisSetAcceptBlockedDriveSignal(nDeCtrlDWord:=Axis1.PlcToNc.ControlDWord , bEnable:=NOT(stAxis1.ctrl.bPositiveLimitSwitch AND stAxis1.ctrl.bNegativeLimitSwitch) ) ;
	
	
(*Set Position *)
	fbSetPosition(
		Axis:= Axis1, 
		Execute:= stAxis1.ctrl.bSetPosition, 
		Position:= stAxis1.ctrl.fSetPosition, 
		Mode:= , 
		Options:= , 
		Done=> stAxis1.stat.bSetPositionDone, 
		Busy=> stAxis1.stat.bSetPositionBusy, 
		Error=> stAxis1.stat.bSetPositionError, 
		ErrorID=> stAxis1.stat.iSetPositionErrID );
	
	
(*Jog *)
	fbJog(
		Axis:= Axis1, 
		JogForward:= stAxis1.ctrl.bJogForward, 
		JogBackwards:= stAxis1.ctrl.bJogBackwards, 
		Mode:= stAxis1.ctrl.eJogMode, 
		Position:= stAxis1.ctrl.fJogPosition, 
		Velocity:= stAxis1.ctrl.fJogVelocity, 
		Acceleration:= stAxis1.ctrl.fJogAcc, 
		Deceleration:= stAxis1.ctrl.fJogDec, 
		Jerk:= , 
		Done=> stAxis1.stat.bJogDone, 
		Busy=> stAxis1.stat.bJogBusy, 
		Active=> stAxis1.stat.bJogActive, 
		CommandAborted=> stAxis1.stat.bJogAborted, 
		Error=> stAxis1.stat.bJogError, 
		ErrorID=> stAxis1.stat.iJogErrID);
	
	
(*Move Relative *)
	fbMoveRelative(
		Axis:= Axis1, 
		Execute:= stAxis1.ctrl.bMoveRelative, 
		Distance:= stAxis1.ctrl.fMoveRelDistance, 
		Velocity:= stAxis1.ctrl.fMoveRelVelocity, 
		Acceleration:= stAxis1.ctrl.fMoveRelAcc,
		Deceleration:= stAxis1.ctrl.fMoveRelDec, 
		Jerk:= , 
		BufferMode:= stAxis1.ctrl.eMoveRelBufferMode, 
		Options:= , 
		Done=> stAxis1.stat.bMoveRelDone, 
		Busy=> stAxis1.stat.bMoveRelBusy, 
		Active=> stAxis1.stat.bMoveRelActive, 
		CommandAborted=> stAxis1.stat.bMoveRelAborted, 
		Error=> stAxis1.stat.bMoveRelErr, 
		ErrorID=> stAxis1.stat.iMoveRelErrID);
		
		
(*Move Absolute *)
	fbMoveAbsolute(
		Axis:= Axis1, 
		Execute:= stAxis1.ctrl.bMoveAbsolute, 
		Position:= stAxis1.ctrl.fMoveAbsPosition, 
		Velocity:= stAxis1.ctrl.fMoveAbsVelocity, 
		Acceleration:= stAxis1.ctrl.fMoveAbsAcc, 
		Deceleration:= stAxis1.ctrl.fMoveAbsDec, 
		Jerk:= , 
		BufferMode:= stAxis1.ctrl.eMoveAbsBufferMode, 
		Options:= , 
		Done=> stAxis1.stat.bMoveAbsDone, 
		Busy=> stAxis1.stat.bMoveAbsBusy, 
		Active=> stAxis1.stat.bMoveAbsActive, 
		CommandAborted=> stAxis1.stat.bMoveAbsAborted, 
		Error=> stAxis1.stat.bMoveAbsErr, 
		ErrorID=> stAxis1.stat.iMoveAbsErrID );
		
	
(*Move Absolute Blending*)
	fbMoveAbsoluteBlending(
		Axis:= Axis1, 
		Execute:= stAxis1.ctrl.bMoveAbsoluteBlending, 
		Position:= stAxis1.ctrl.fMoveAbsBlendingPosition, 
		Velocity:= stAxis1.ctrl.fMoveAbsBlendingAcc, 
		Acceleration:= stAxis1.ctrl.fMoveAbsBlendingAcc, 
		Deceleration:= stAxis1.ctrl.fMoveAbsBlendingDec, 
		Jerk:= , 
		BufferMode:= stAxis1.ctrl.eMoveAbsBlendingBufferMode, 
		Options:= , 
		Done=> stAxis1.stat.bMoveAbsBlendingDone, 
		Busy=> stAxis1.stat.bMoveAbsBlendingBusy, 
		Active=> stAxis1.stat.bMoveAbsBlendingActive, 
		CommandAborted=> stAxis1.stat.bMoveAbsBlendingAborted, 
		Error=> stAxis1.stat.bMoveAbsBlendingErr, 
		ErrorID=> stAxis1.stat.iMoveAbsBlendingErrID );	
		
		
(*Move Modulo *)
	fbMoveModulo(
		Axis:= Axis1, 
		Execute:= stAxis1.ctrl.bMoveModulo, 
		Position:= stAxis1.ctrl.fMoveModuloPosition, 
		Velocity:= stAxis1.ctrl.fMoveModuloVelocity, 
		Acceleration:= stAxis1.ctrl.fMoveModuloAcc, 
		Deceleration:= stAxis1.ctrl.fMoveModuloDec, 
		Jerk:= , 
		Direction:= stAxis1.ctrl.eMoveModuloDirection, 
		BufferMode:= stAxis1.ctrl.eMoveModuloBufferMode, 
		Options:= , 
		Done=> stAxis1.stat.bMoveModuloDone, 
		Busy=> stAxis1.stat.bMoveModuloBusy, 
		Active=> stAxis1.stat.bMoveModuloActive, 
		CommandAborted=> stAxis1.stat.bMoveModuloAborted, 
		Error=> stAxis1.stat.bMoveModuloErr, 
		ErrorID=> stAxis1.stat.iMoveModuloErrID);		
			
		
(*Move Velocity*)	
		
	ReMoveVelocity(CLK:= stAxis1.ctrl.bMoveVelocity, Q=> );
	FeMoveVelocity(CLK:= stAxis1.ctrl.bMoveVelocity, Q=> );

	
	bMoveVelocity	:=	ReMoveVelocity.Q
						OR (
								(stAxis1.ctrl.bMoveVelocity AND (stAxis1.ctrl.fMoveVelVelocity<>oldMoveVeloVelocity))
								OR (stAxis1.ctrl.bMoveVelocity AND (stAxis1.ctrl.eMoveVelDirection<>oldDirection))
							);
							
	fbMoveVelocity(
		Axis:= Axis1, 
		Execute:= bMoveVelocity, 
		Velocity:= stAxis1.ctrl.fMoveVelVelocity, 
		Acceleration:= stAxis1.ctrl.fMoveVelAcc, 
		Deceleration:= stAxis1.ctrl.fMoveVelDec, 
		Jerk:= , 
		Direction:=stAxis1.ctrl.eMoveVelDirection , 
		BufferMode:= stAxis1.ctrl.eMoveVelBufferMode, 
		Options:= , 
		InVelocity=> stAxis1.stat.bMoveVeloInVelocity, 
		Busy=> stAxis1.stat.bMoveVeloBusy, 
		Active=> stAxis1.stat.bMoveVeloActive, 
		CommandAborted=> stAxis1.stat.bMoveVeloAborted, 
		Error=> stAxis1.stat.bMoveVeloErr, 
		ErrorID=> stAxis1.stat.iMoveVeloErrID);		
		
	oldMoveVeloVelocity:=stAxis1.ctrl.fMoveVelVelocity;
	oldDirection:=stAxis1.ctrl.eMoveVelDirection;
		
		
(*Positional Stop *)	

	bStopAxis1:=(FeMoveVelocity.Q OR stAxis1.ctrl.bStopAxis);

	fbMoveVeloPosStop(
		Axis:= Axis1, 
		Execute:= (bStopAxis1 AND stAxis1.ctrl.bMoveVelPositionalStopEnable), 
		Position:= stAxis1.ctrl.fMoveVelPositionalStopPos, 
		Velocity:= stAxis1.ctrl.fMoveVelVelocity, 
		Acceleration:= stAxis1.ctrl.fMoveVelPositionalStopAcc, 
		Deceleration:= stAxis1.ctrl.fMoveVelPositionalStopDec, 
		Jerk:= , 
		BufferMode:= stAxis1.ctrl.eMoveVelPositionalStopBufferMode, 
		Options:= , 
		Done=> stAxis1.stat.bMoveVeloPosStopDone, 
		Busy=> stAxis1.stat.bMoveVeloPosStopBusy, 
		Active=> stAxis1.stat.bMoveVeloPosStopActive, 
		CommandAborted=> stAxis1.stat.bMoveVeloPosStopAborted, 
		Error=> stAxis1.stat.bMoveVeloPosStopErr, 
		ErrorID=> stAxis1.stat.iMoveVeloPosStopErrID);
	

(*Gear In Dynamic *)		
	fbGearInDyn(
		Master:= Axis1, 
		Slave:= SlaveAxis, 
		Enable:= stAxis1.ctrl.bGearInDynamic, 
		GearRatio:= stAxis1.ctrl.fGearInDynRatio, 
		Acceleration:= stAxis1.ctrl.fGearInDynAcc, 
		Deceleration:= stAxis1.ctrl.fGearInDynDec, 
		Jerk:= , 
		BufferMode:= , 
		Options:= , 
		InGear=> stAxis1.stat.bGearInDynInGear, 
		Busy=> stAxis1.stat.bGearInDynBusy, 
		Active=> stAxis1.stat.bGearInDynActive, 
		CommandAborted=> stAxis1.stat.bGearInDynAborted, 
		Error=> stAxis1.stat.bGearInDynErr, 
		ErrorID=> stAxis1.stat.iGearInDynErrID);


(*Gear In Dynamic Axis1 to Master *)		
	fbGearInDyn_Axis1toMaster(
		Master:= MasterAxis, 
		Slave:= Axis1, 
		Enable:= stAxis1.ctrl.bGearInDynamic_Axis1toMaster, 
		GearRatio:= stAxis1.ctrl.fGearInDynRatio_Axis1toMaster, 
		Acceleration:= stAxis1.ctrl.fGearInDynAcc_Axis1toMaster, 
		Deceleration:= stAxis1.ctrl.fGearInDynDec_Axis1toMaster, 
		Jerk:= , 
		BufferMode:= , 
		Options:= , 
		InGear=> stAxis1.stat.bGearInDynInGear_Axis1toMaster, 
		Busy=> stAxis1.stat.bGearInDynBusy_Axis1toMaster, 
		Active=> stAxis1.stat.bGearInDynActive_Axis1toMaster, 
		CommandAborted=> stAxis1.stat.bGearInDynAborted_Axis1toMaster, 
		Error=> stAxis1.stat.bGearInDynErr_Axis1toMaster, 
		ErrorID=> stAxis1.stat.iGearInDynErrID_Axis1toMaster);
	
		
(*Gear In Multi Master *)		
	fbGearInMultiMaster(
		Master1:= Axis1, 
		Master2:= Axis2, 
		Master3:= Axis3, 
		Master4:= Axis4, 
		Slave:= SlaveAxis, 
		Enable:= stAxis1.ctrl.bGearInMultimaster, 
		GearRatio1:= stAxis1.ctrl.fGearRatioMaster1, 
		GearRatio2:= stAxis1.ctrl.fGearRatioMaster2, 
		GearRatio3:= stAxis1.ctrl.fGearRatioMaster3, 
		GearRatio4:= stAxis1.ctrl.fGearRatioMaster4, 
		Acceleration:= stAxis1.ctrl.fGearInMultimasterAcc, 
		Deceleration:= stAxis1.ctrl.fGearInMultimasterDec, 
		Jerk:= , 
		BufferMode:= , 
		Options:= , 
		InGear=> stAxis1.stat.bGearInMultimasterInGear, 
		Busy=> stAxis1.stat.bGearInMultimasterBusy, 
		Active=> stAxis1.stat.bGearInMultimasterActive, 
		CommandAborted=> stAxis1.stat.bGearInMultimasterAborted, 
		Error=> stAxis1.stat.bGearInMultimasterErr, 
		ErrorID=> stAxis1.stat.iGearInMultimasterGrErrID);	
	
		
(*Move Superimposed *)		
	fbMoveSuperImposed(
		Axis:= SlaveAxis, 
		Execute:= stAxis1.ctrl.bMoveSuperimposed, 
		Mode:= stAxis1.ctrl.eMoveSupImpMode, 
		Distance:= stAxis1.ctrl.fMoveSupImpDistance, 
		VelocityDiff:= stAxis1.ctrl.fMoveSupImpVelocityDiff, 
		Acceleration:= stAxis1.ctrl.fMoveSupImpAcc, 
		Deceleration:= stAxis1.ctrl.fMoveSupImpDec, 
		Jerk:= , 
		VelocityProcess:= stAxis1.ctrl.fMoveSupImpVelocityProcess, 
		Length:= stAxis1.ctrl.fMoveSupImpLength, 
		Options:= stAxis1.ctrl.eMoveSupImpOptions, 
		Done=> stAxis1.stat.bMoveSupImpDone, 
		Busy=> stAxis1.stat.bMoveSupImpBusy, 
		Active=> stAxis1.stat.bMoveSupImpActive, 
		CommandAborted=> stAxis1.stat.bMoveSupImpAborted, 
		Error=> stAxis1.stat.bMoveSupImpErr, 
		ErrorID=> stAxis1.stat.iMoveSupImpErrorId, 
		Warning=> stAxis1.stat.bMoveSupImpWarning, 
		WarningId=> stAxis1.stat.iMoveSupImpWarningID, 
		ActualVelocityDiff=> stAxis1.stat.fMoveSupImpActualVelocityDiff, 
		ActualDistance=> stAxis1.stat.fMoveSupImpActualDistance, 
		ActualLength=> stAxis1.stat.fMoveSupImpActualLength, 
		ActualAcceleration=> stAxis1.stat.fMoveSupImpActualAcc, 
		ActualDeceleration=> stAxis1.stat.fMoveSupImpActualDec );		
			
					
(*Gear Out *)	
	fbGearOut(
		Slave:= SlaveAxis, 
		Execute:= stAxis1.ctrl.bGearOutSlaveAxis, 
		Options:= , 
		Done=> stAxis1.stat.bGearOutSlaveAxisDone, 
		Busy=> stAxis1.stat.bGearOutSlaveAxisBusy, 
		Error=> stAxis1.stat.bGearOutSlaveAxisErr, 
		ErrorID=> stAxis1.stat.iGearOutSlaveAxisErrID );	

		
(*Gear Out Axis1 from Master*)	
	fbGearOutAxis1fromMaster(
		Slave:= SlaveAxis, 
		Execute:= stAxis1.ctrl.bGearOutAxis1fromMaster, 
		Options:= , 
		Done=> stAxis1.stat.bGearOutAxis1fromMasterDone, 
		Busy=> stAxis1.stat.bGearOutAxis1fromMasterBusy, 
		Error=> stAxis1.stat.bGearOutAxis1fromMasterErr, 
		ErrorID=> stAxis1.stat.iGearOutAxis1fromMasterErrID );			
		

(*Stop SlaveAxis *)
	fbStopSlave(
		Axis:= SlaveAxis, 
		Execute:= stAxis1.stat.bGearOutSlaveAxisDone, 
		Deceleration:= , 
		Jerk:= , 
		Options:= , 
		Done=> stAxis1.stat.bStopSlaveAxisDone, 
		Busy=> stAxis1.stat.bStopSlaveAxisBusy, 
		Active=> stAxis1.stat.bStopSlaveAxisActive, 
		CommandAborted=> stAxis1.stat.bStopSlaveAxisAborted, 
		Error=> stAxis1.stat.bStopSlaveAxisErr, 
		ErrorID=> stAxis1.stat.iStopSlaveAxisErrorID );


(*Touch Probe*)
	fbTouchProbe(
		Axis:= Axis1, 
		TriggerInput:= stAxis1.ctrl.eTouchProbeTriggerRef, 
		Execute:= stAxis1.ctrl.bTouchProbe, 
		WindowOnly:= stAxis1.ctrl.bTouchProbeWindowOnly, 
		FirstPosition:= stAxis1.ctrl.fTouchProbeFirstPosition, 
		LastPosition:= stAxis1.ctrl.fTouchProbeLastPosition, 
		Done=> stAxis1.stat.bTouchProbeDone, 
		Busy=> stAxis1.stat.bTouchProbeBusy, 
		CommandAborted=> stAxis1.stat.bTouchProbeAborted, 
		Error=> stAxis1.stat.bTouchProbeErr, 
		ErrorID=> stAxis1.stat.iTouchProbeErrID, 
		RecordedPosition=> stAxis1.stat.fTouchProbeRecordedPosition);


(*Abort Trigger*)	
	fbAbortTrigger(
		Axis:= Axis1, 
		TriggerInput:= stAxis1.ctrl.eTouchProbeTriggerRef, 
		Execute:= stAxis1.ctrl.bTouchProbeAbortTrigger, 
		Done=> stAxis1.stat.bAbortTouchProbeDone, 
		Busy=> stAxis1.stat.bAbortTouchProbeBusy, 
		Error=> stAxis1.stat.bAbortTouchProbeErr, 
		ErrorID=> stAxis1.stat.iAbortTouchProbeErrID );	
		
		
(*Stop Axis1 *)
		fbStopMaster(
			Axis:= Axis1, 
			Execute:= (stAxis1.ctrl.bStopAxis OR FeMoveVelocity.Q OR stAxis1.stat.bGearOutAxis1fromMasterDone), 
			Deceleration:= stAxis1.ctrl.fStopAxisDec, 
			Jerk:= , 
			Options:= , 
			Done=> stAxis1.stat.bStopAxisDone, 
			Busy=> stAxis1.stat.bStopAxisBusy, 
			Active=> stAxis1.stat.bStopAxisActive, 
			CommandAborted=> stAxis1.stat.bStopAxisAborted, 
			Error=> stAxis1.stat.bStopAxisErr, 
			ErrorID=> stAxis1.stat.iStopAxisErrID );
		
			
			
			
(*External Setposition Generation ****************************************************)

	CASE ExtSP_State OF
	
		0:
			stAxis1.stat.bExtSetPositionDone:=FALSE;
			stAxis1.stat.bExtSetPositionBusy:=FALSE;
			stAxis1.stat.bExtSetPositionErr:=FALSE;
			stAxis1.stat.iExtSetPositionErrID:=0;
			
			IF stAxis1.ctrl.bExtSetPointGenEnable THEN
				stAxis1.stat.bExtSetPositionBusy:=TRUE;
				preExtSP_State:=ExtSP_State;
				ExtSP_State:=10;
			END_IF
	
	
		10:(*ExtSetPointGenEnable*)
			IF stAxis1.ctrl.bExtSetPointGenEnable THEN
	
				fbExtSetPointGenEnable(
					Execute:=TRUE ,
					Position:= ,
					PositionType:=stAxis1.ctrl.eExtSetPositionType ,
					Axis:=Axis1 ,
					Done=> ,
					Busy=> ,
					Error=> ,
					ErrorID=> , 
					Enabled=> );
	
				IF NOT(fbExtSetPointGenEnable.Error) THEN
					IF fbExtSetPointGenEnable.Done THEN
	
						fbExtSetPointGenEnable(
							Execute:=FALSE ,
							Position:= ,
							PositionType:=stAxis1.ctrl.eExtSetPositionType ,
							Axis:=Axis1 ,
							Done=> ,
							Busy=> ,
							Error=> ,
							ErrorID=> , 
							Enabled=> );
		
						preExtSP_State:=ExtSP_State;
						ExtSP_State:=100;
	
					END_IF
				ELSE
					stAxis1.stat.bExtSetPositionErr:=TRUE;
					stAxis1.stat.iExtSetPositionErrID:=fbExtSetPointGenEnable.ErrorID;
					preExtSP_State:=ExtSP_State;
					ExtSP_State:=999;
				END_IF
	
			ELSE
				preExtSP_State:=ExtSP_State;
				ExtSP_State:=800;
			END_IF
	
	
		100:
			IF stAxis1.ctrl.bExtSetPointGenEnable THEN
	
				stAxis1.stat.bExtSetPositionReady:=TRUE;
	
			ELSE
				stAxis1.stat.bExtSetPositionReady:=FALSE;
				preExtSP_State:=ExtSP_State;
				ExtSP_State:=800;
			END_IF
	
	
	
		800:(*ExtSetPointGenDisable*)
			fbExtSetPointGenEnable(
				Execute:=FALSE ,
				Position:= ,
				PositionType:=stAxis1.ctrl.eExtSetPositionType ,
				Axis:=Axis1 ,
				Done=> ,
				Busy=> ,
				Error=> ,
				ErrorID=> , 
				Enabled=> );
	
			IF NOT(fbExtSetPointGenEnable.Busy) THEN
				preExtSP_State:=ExtSP_State;
				ExtSP_State:=810;
			END_IF
	
	
		810:
	
			fbExtSetPointGenDisable(
				Execute:=TRUE ,
				Axis:=Axis1 ,
				Done=> ,
				Busy=> , 
				Error=> , 
				ErrorID=> , 
				Enabled=> );
	
			IF NOT(fbExtSetPointGenDisable.Error) THEN
				IF fbExtSetPointGenDisable.Done THEN
					fbExtSetPointGenDisable(
						Execute:=FALSE ,
						Axis:=Axis1 ,
						Done=> ,
						Busy=> , 
						Error=> , 
						ErrorID=> , 
						Enabled=> );
	
					stAxis1.stat.bExtSetPositionDone:=TRUE;
	
					preExtSP_State:=ExtSP_State;
					ExtSP_State:=0;
	
				END_IF
			ELSE
				stAxis1.stat.bExtSetPositionErr:=TRUE;
				stAxis1.stat.iExtSetPositionErrID:=fbExtSetPointGenDisable.ErrorID;
				preExtSP_State:=ExtSP_State;
				ExtSP_State:=999;
			END_IF
	
	
	
		999:(*ExtSetPointGen Error*)
	
			fbExtSetPointGenEnable(
				Execute:=FALSE ,
				Position:= ,
				PositionType:=stAxis1.ctrl.eExtSetPositionType ,
				Axis:=Axis1 ,
				Done=> ,
				Busy=> ,
				Error=> ,
				ErrorID=> , 
				Enabled=> );
	
			fbExtSetPointGenDisable(
				Execute:=FALSE ,
				Axis:=Axis1 ,
				Done=> ,
				Busy=> , 
				Error=> , 
				ErrorID=> , 
				Enabled=> );
	
	
			IF NOT(stAxis1.ctrl.bExtSetPointGenEnable) THEN
				stAxis1.stat.bExtSetPositionErr:=FALSE;
				preExtSP_State:=ExtSP_State;
				ExtSP_State:=0;
			END_IF
	
	END_CASE
	

(*Position Feed*)
	MC_ExtSetPointGenFeed(
		Position:=stAxis1.ctrl.fExtSetPosition,
		Velocity:=stAxis1.ctrl.fExtSetVelocity,
		Acceleration:=stAxis1.ctrl.fExtSetAcceleration,
		Direction:=stAxis1.ctrl.iExtSetDirection,
		Axis:=Axis1);
	
(*External Setposition Generation ///////////////////////////////////////////////////*)
			
			
			
			
			
			
			
END_FUNCTION_BLOCK
